FUNCTION_BLOCK FB_LamparaConmutada_LD
VAR_INPUT
END_VAR
VAR_OUTPUT
END_VAR
VAR
    Lampara AT %Q*: BOOL;
    Pulsador AT %I*: BOOL;
    MemoriaLampara: BOOL;
    
    Pulsacion: R_TRIG;
END_VAR

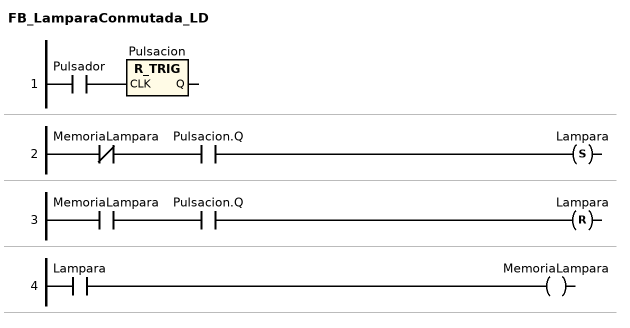
// NETWORK 1
Pulsacion(CLK := Pulsador); // R_TRIG

// NETWORK 2
Lampara S= NOT MemoriaLampara AND Pulsacion.Q;

// NETWORK 3
Lampara R= MemoriaLampara AND Pulsacion.Q;

// NETWORK 4
MemoriaLampara := Lampara;

END_FUNCTION_BLOCK

(* stored: Version 1.1.0.1, ProductVersion 3.1.4024.12
   POU FB_LamparaConmutada_LD: Id {fb9e8f1e-35ac-4616-995f-8d9dee686820}, SpecialFunc None *)
